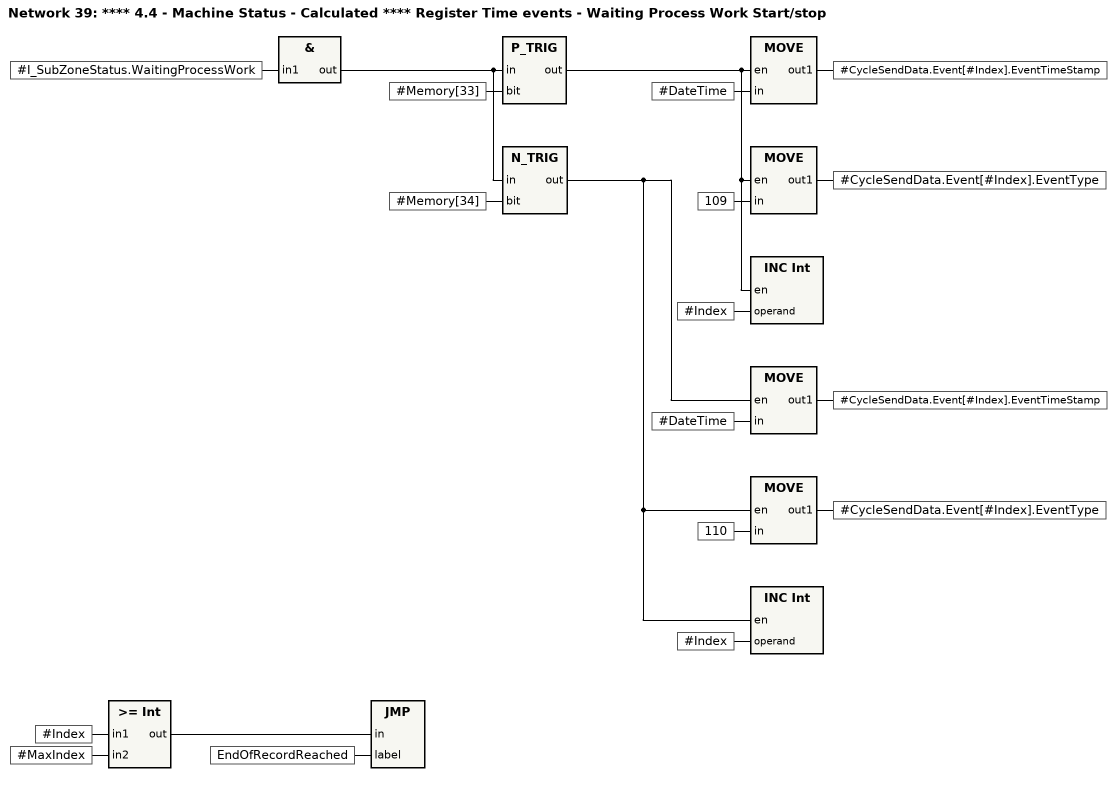
   #_w1 := #I_SubZoneStatus.WaitingProcessWork AND NOT #Memory[33];   // rising edge
   #Memory[33] := #I_SubZoneStatus.WaitingProcessWork;
   IF #_w1 THEN
       #CycleSendData.Event[#Index].EventTimeStamp := #DateTime;
       #CycleSendData.Event[#Index].EventType := 109;
       #Index := #Index + 1;
   END_IF;
   #_w2 := NOT #I_SubZoneStatus.WaitingProcessWork AND #Memory[34];   // falling edge
   #Memory[34] := #I_SubZoneStatus.WaitingProcessWork;
   IF #_w2 THEN
       #CycleSendData.Event[#Index].EventTimeStamp := #DateTime;
       #CycleSendData.Event[#Index].EventType := 110;
       #Index := #Index + 1;
   END_IF;
   IF #Index >= #MaxIndex THEN GOTO EndOfRecordReached; END_IF;
END_REGION

REGION Network 40: **** 4.4 - Machine Status - Calculated **** Register Time events - Process Work Start/stop
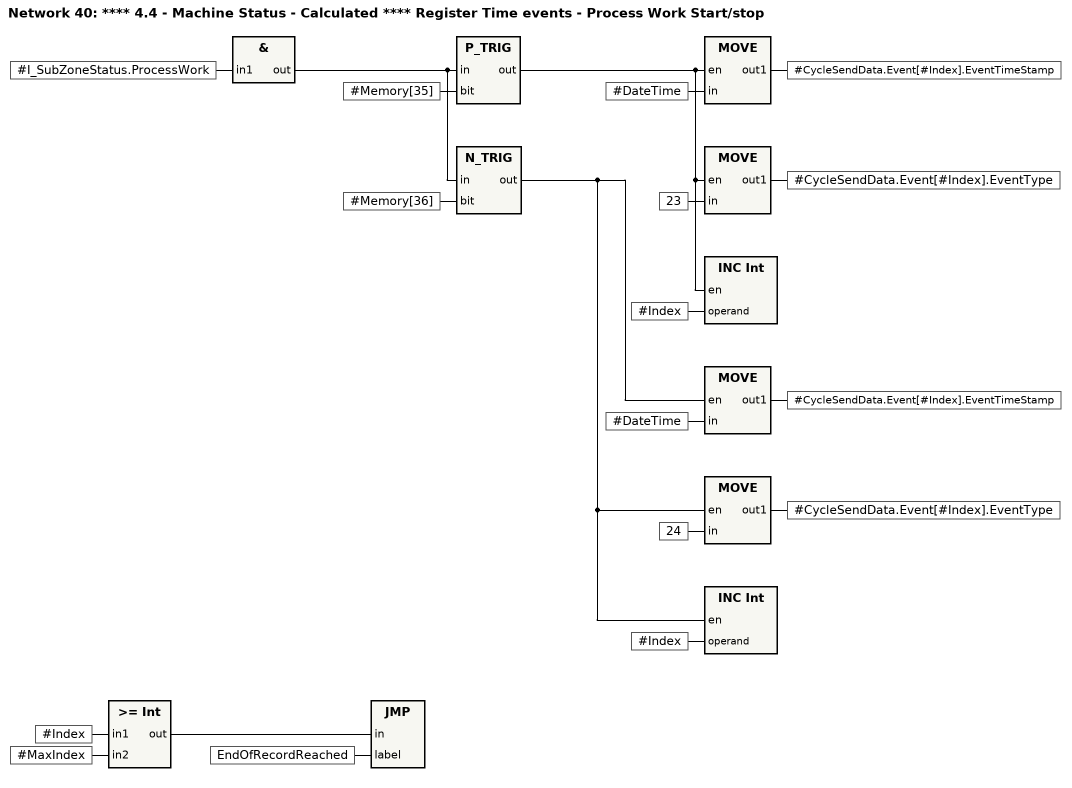
   #_w1 := #I_SubZoneStatus.ProcessWork AND NOT #Memory[35];   // rising edge
   #Memory[35] := #I_SubZoneStatus.ProcessWork;
   IF #_w1 THEN
       #CycleSendData.Event[#Index].EventTimeStamp := #DateTime;
       #CycleSendData.Event[#Index].EventType := 23;
       #Index := #Index + 1;
   END_IF;
   #_w2 := NOT #I_SubZoneStatus.ProcessWork AND #Memory[36];   // falling edge
   #Memory[36] := #I_SubZoneStatus.ProcessWork;
   IF #_w2 THEN
       #CycleSendData.Event[#Index].EventTimeStamp := #DateTime;
       #CycleSendData.Event[#Index].EventType := 24;
       #Index := #Index + 1;
   END_IF;
   IF #Index >= #MaxIndex THEN GOTO EndOfRecordReached; END_IF;
END_REGION

REGION Network 41: **** 4.4 - Machine Status - Calculated **** Register Time events - Cycle Hold
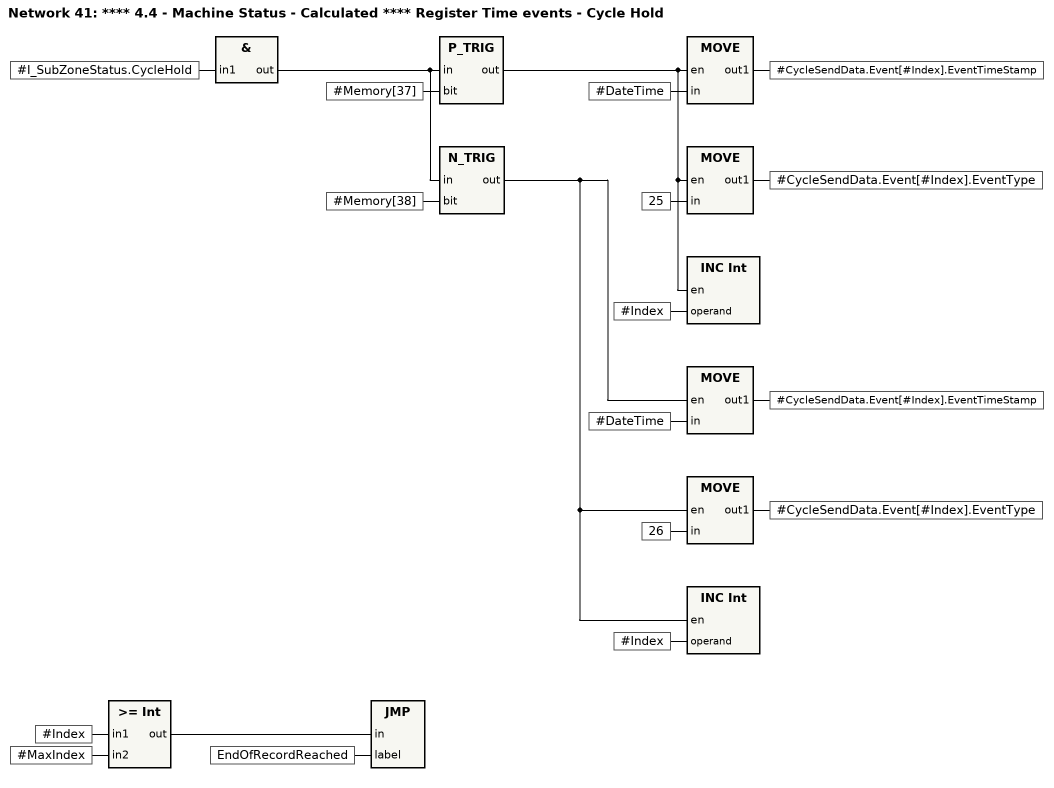
   #_w1 := #I_SubZoneStatus.CycleHold AND NOT #Memory[37];   // rising edge
   #Memory[37] := #I_SubZoneStatus.CycleHold;
   IF #_w1 THEN
       #CycleSendData.Event[#Index].EventTimeStamp := #DateTime;
       #CycleSendData.Event[#Index].EventType := 25;
       #Index := #Index + 1;
   END_IF;
   #_w2 := NOT #I_SubZoneStatus.CycleHold AND #Memory[38];   // falling edge
   #Memory[38] := #I_SubZoneStatus.CycleHold;
   IF #_w2 THEN
       #CycleSendData.Event[#Index].EventTimeStamp := #DateTime;
       #CycleSendData.Event[#Index].EventType := 26;
       #Index := #Index + 1;
   END_IF;
   IF #Index >= #MaxIndex THEN GOTO EndOfRecordReached; END_IF;
END_REGION

REGION Network 42: **** 4.4 - Machine Status - Calculated **** Register Time events - WaitingOutput1 Start/stop
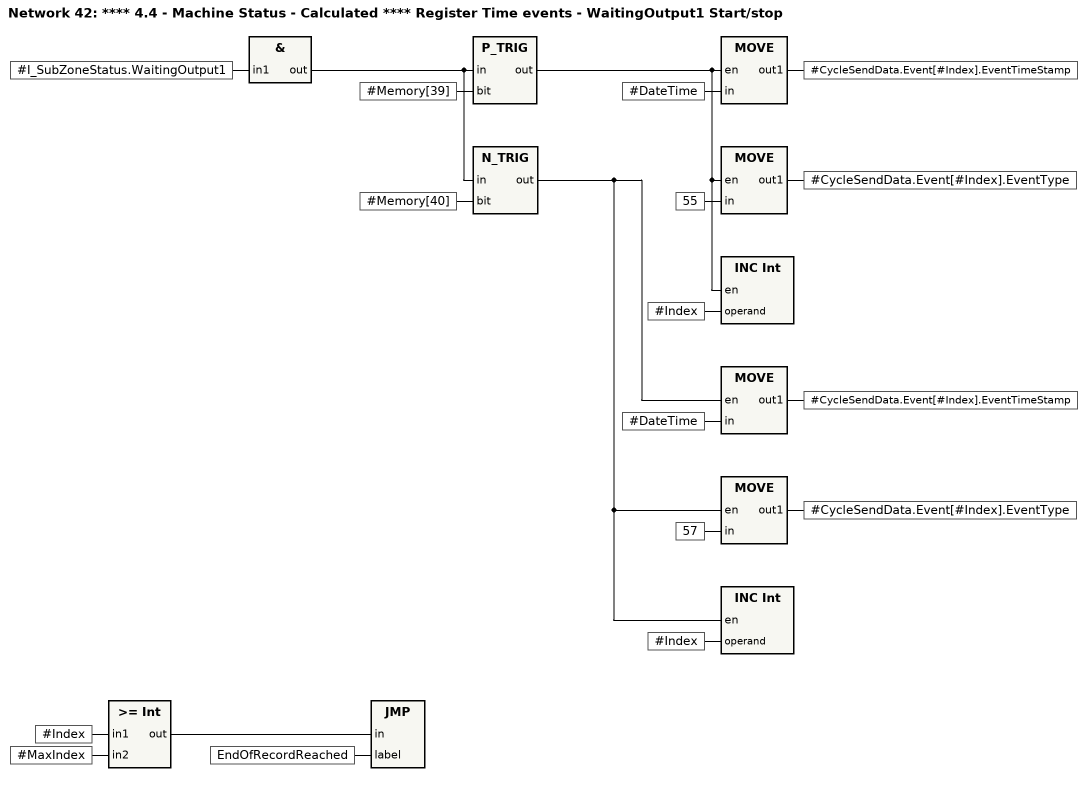
   #_w1 := #I_SubZoneStatus.WaitingOutput1 AND NOT #Memory[39];   // rising edge
   #Memory[39] := #I_SubZoneStatus.WaitingOutput1;
   IF #_w1 THEN
       #CycleSendData.Event[#Index].EventTimeStamp := #DateTime;
       #CycleSendData.Event[#Index].EventType := 55;
       #Index := #Index + 1;
   END_IF;
   #_w2 := NOT #I_SubZoneStatus.WaitingOutput1 AND #Memory[40];   // falling edge
   #Memory[40] := #I_SubZoneStatus.WaitingOutput1;
   IF #_w2 THEN
       #CycleSendData.Event[#Index].EventTimeStamp := #DateTime;
       #CycleSendData.Event[#Index].EventType := 57;
       #Index := #Index + 1;
   END_IF;
   IF #Index >= #MaxIndex THEN GOTO EndOfRecordReached; END_IF;
END_REGION

REGION Network 43: **** 4.4 - Machine Status - Calculated **** Register Time events - WaitingOutput2 Start/stop
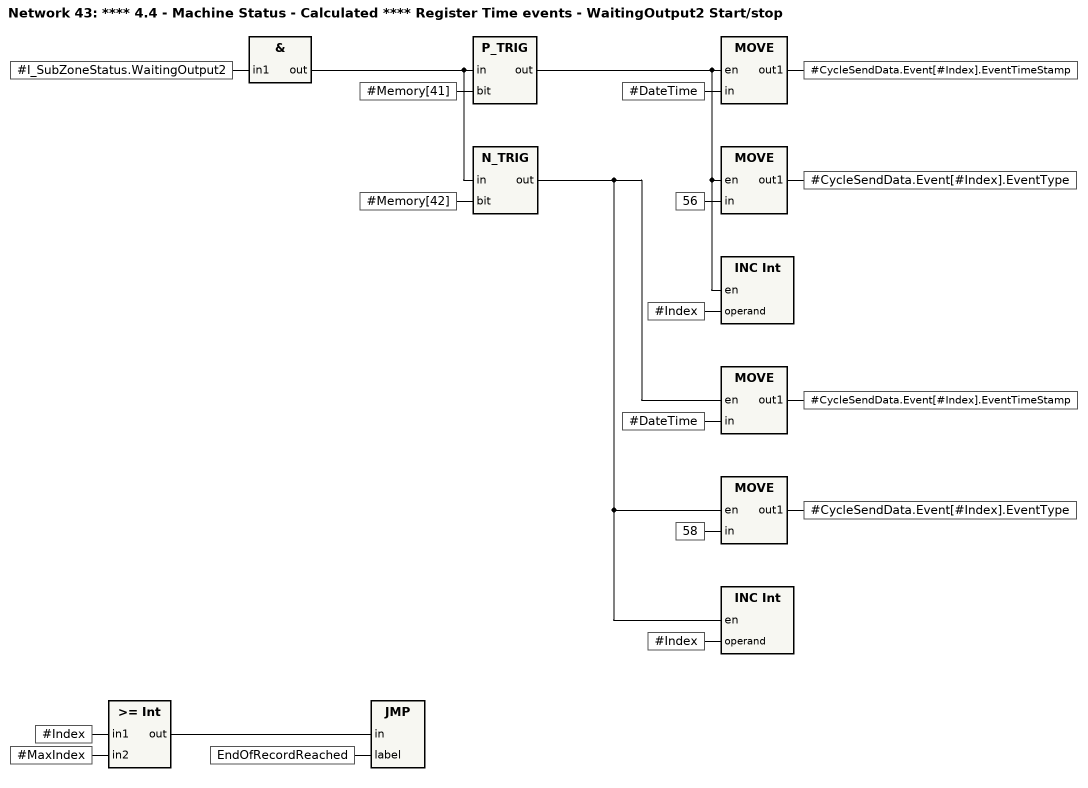
   #_w1 := #I_SubZoneStatus.WaitingOutput2 AND NOT #Memory[41];   // rising edge
   #Memory[41] := #I_SubZoneStatus.WaitingOutput2;
   IF #_w1 THEN
       #CycleSendData.Event[#Index].EventTimeStamp := #DateTime;
       #CycleSendData.Event[#Index].EventType := 56;
       #Index := #Index + 1;
   END_IF;
   #_w2 := NOT #I_SubZoneStatus.WaitingOutput2 AND #Memory[42];   // falling edge
   #Memory[42] := #I_SubZoneStatus.WaitingOutput2;
   IF #_w2 THEN
       #CycleSendData.Event[#Index].EventTimeStamp := #DateTime;
       #CycleSendData.Event[#Index].EventType := 58;
       #Index := #Index + 1;
   END_IF;
   IF #Index >= #MaxIndex THEN GOTO EndOfRecordReached; END_IF;
END_REGION

REGION Network 44: **** 4.4 - Machine Status - Calculated **** Register Time events - Outfeed1 Start/stop
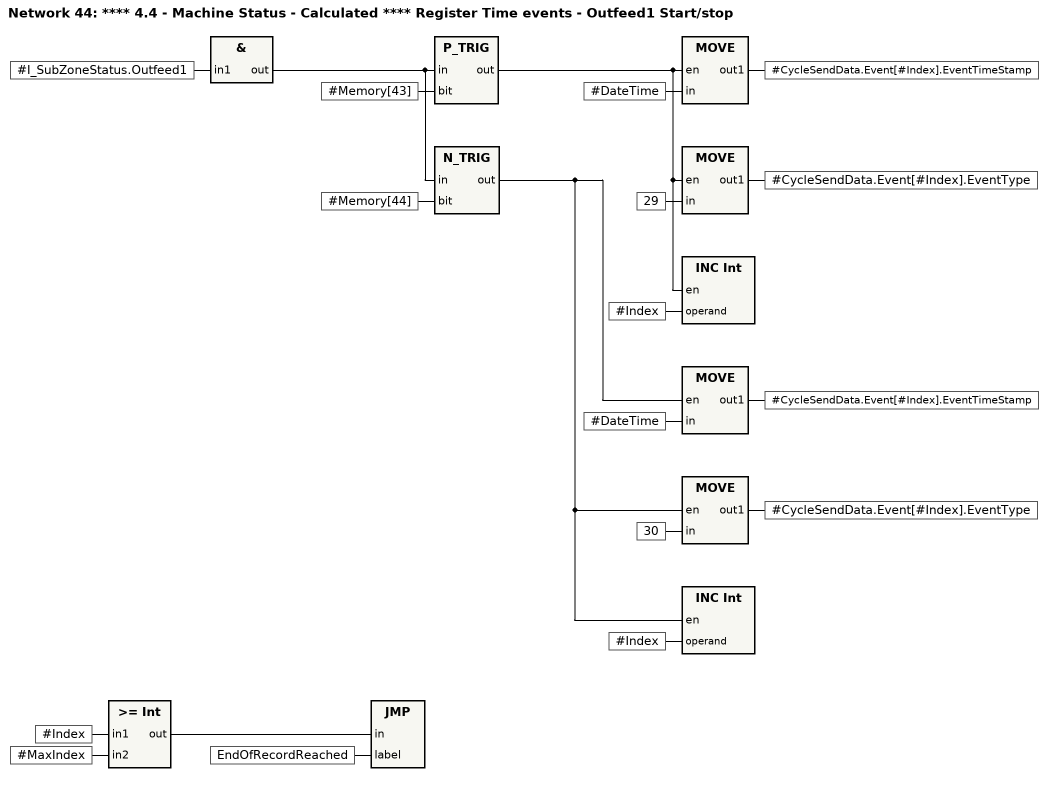
   #_w1 := #I_SubZoneStatus.Outfeed1 AND NOT #Memory[43];   // rising edge
   #Memory[43] := #I_SubZoneStatus.Outfeed1;
   IF #_w1 THEN
       #CycleSendData.Event[#Index].EventTimeStamp := #DateTime;
       #CycleSendData.Event[#Index].EventType := 29;
       #Index := #Index + 1;
   END_IF;
   #_w2 := NOT #I_SubZoneStatus.Outfeed1 AND #Memory[44];   // falling edge
   #Memory[44] := #I_SubZoneStatus.Outfeed1;
   IF #_w2 THEN
       #CycleSendData.Event[#Index].EventTimeStamp := #DateTime;
       #CycleSendData.Event[#Index].EventType := 30;
       #Index := #Index + 1;
   END_IF;
   IF #Index >= #MaxIndex THEN GOTO EndOfRecordReached; END_IF;
END_REGION

REGION Network 45: **** 4.4 - Machine Status - Calculated **** Register Time events - Outfeed2 Start/stop
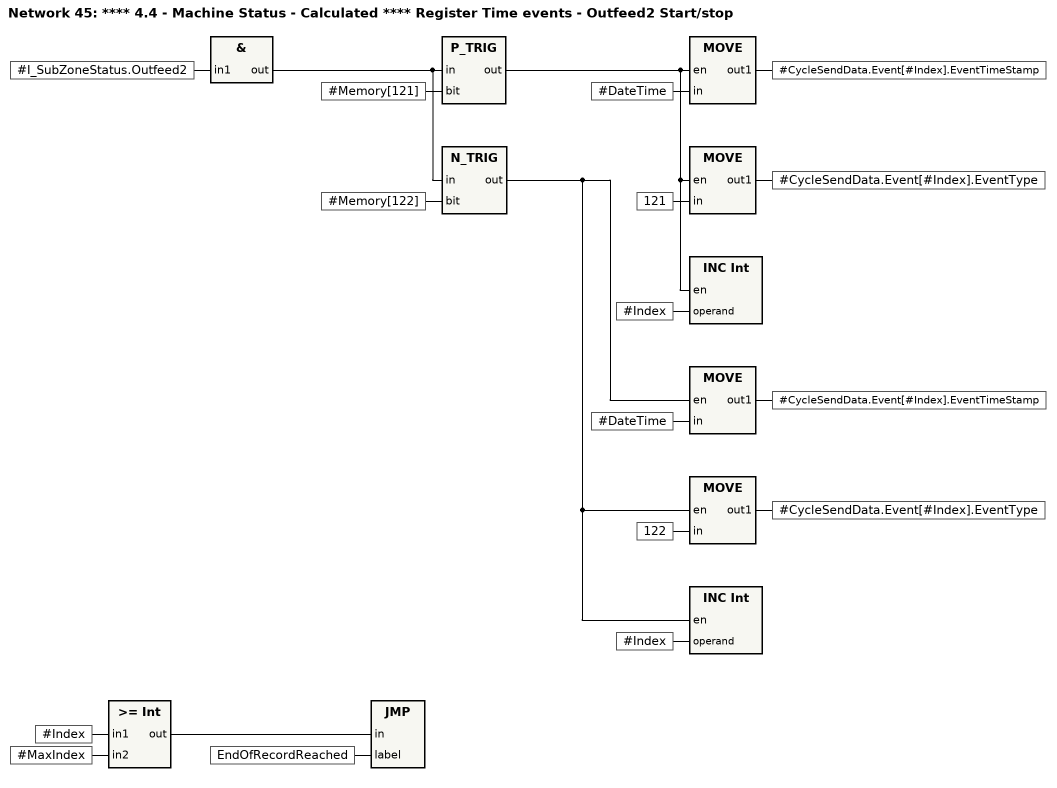
   #_w1 := #I_SubZoneStatus.Outfeed2 AND NOT #Memory[121];   // rising edge
   #Memory[121] := #I_SubZoneStatus.Outfeed2;
   IF #_w1 THEN
       #CycleSendData.Event[#Index].EventTimeStamp := #DateTime;
       #CycleSendData.Event[#Index].EventType := 121;
       #Index := #Index + 1;
   END_IF;
   #_w2 := NOT #I_SubZoneStatus.Outfeed2 AND #Memory[122];   // falling edge
   #Memory[122] := #I_SubZoneStatus.Outfeed2;
   IF #_w2 THEN
       #CycleSendData.Event[#Index].EventTimeStamp := #DateTime;
       #CycleSendData.Event[#Index].EventType := 122;
       #Index := #Index + 1;
   END_IF;
   IF #Index >= #MaxIndex THEN GOTO EndOfRecordReached; END_IF;
END_REGION

REGION Network 46: **** 4.4 - Machine Status - Calculated **** Register Time events - Recovery Time Start/stop
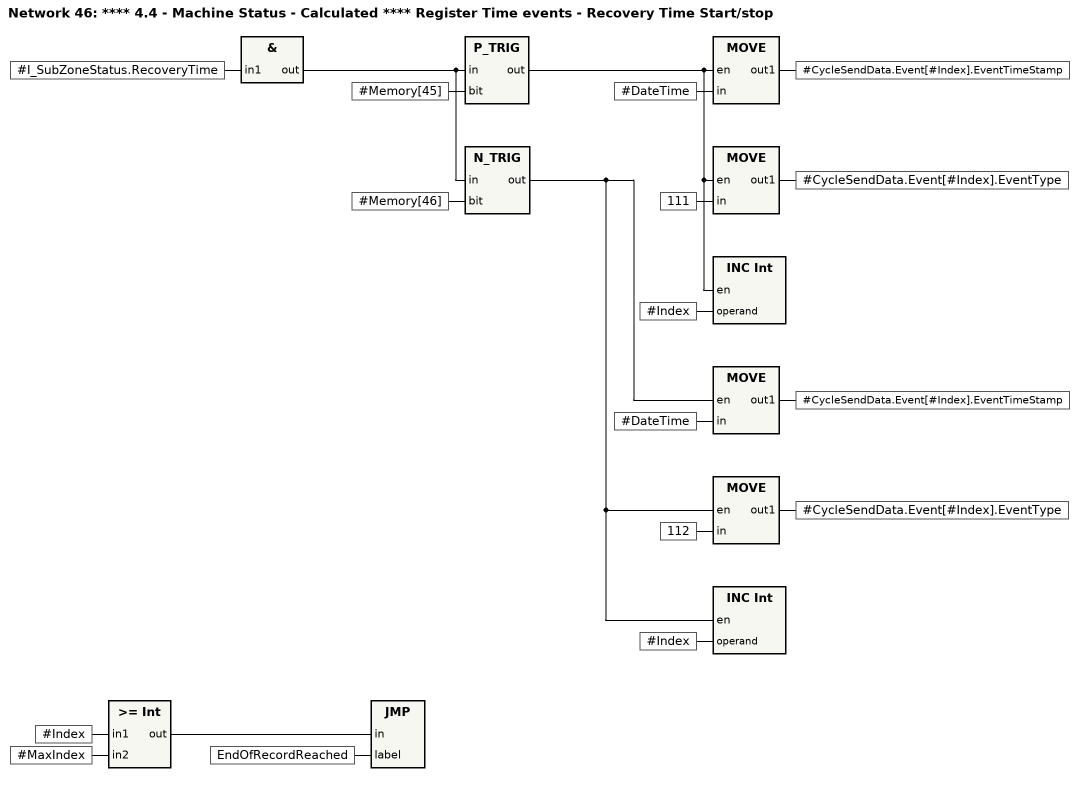
   #_w1 := #I_SubZoneStatus.RecoveryTime AND NOT #Memory[45];   // rising edge
   #Memory[45] := #I_SubZoneStatus.RecoveryTime;
   IF #_w1 THEN
       #CycleSendData.Event[#Index].EventTimeStamp := #DateTime;
       #CycleSendData.Event[#Index].EventType := 111;
       #Index := #Index + 1;
   END_IF;
   #_w2 := NOT #I_SubZoneStatus.RecoveryTime AND #Memory[46];   // falling edge
   #Memory[46] := #I_SubZoneStatus.RecoveryTime;
   IF #_w2 THEN
       #CycleSendData.Event[#Index].EventTimeStamp := #DateTime;
       #CycleSendData.Event[#Index].EventType := 112;
       #Index := #Index + 1;
   END_IF;
   IF #Index >= #MaxIndex THEN GOTO EndOfRecordReached; END_IF;
END_REGION

REGION Network 47: **** 4.4 - Machine Status - Calculated **** Register Time events - QualityNok Start/stop
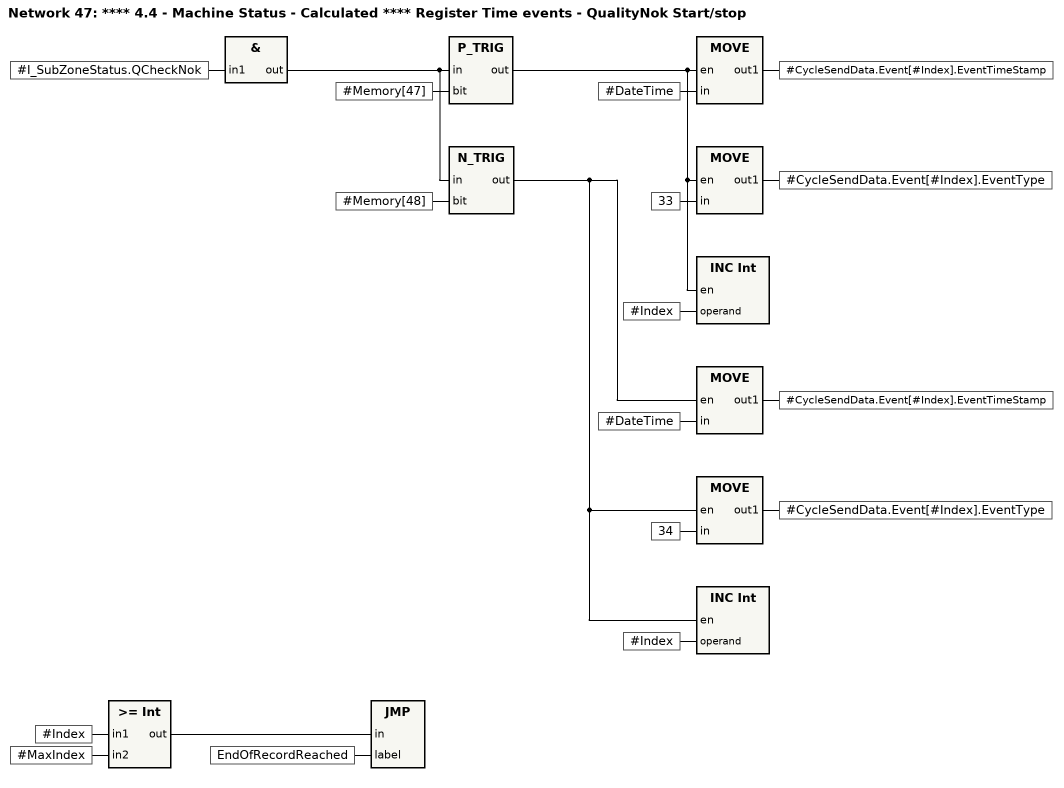
   #_w1 := #I_SubZoneStatus.QCheckNok AND NOT #Memory[47];   // rising edge
   #Memory[47] := #I_SubZoneStatus.QCheckNok;
   IF #_w1 THEN
       #CycleSendData.Event[#Index].EventTimeStamp := #DateTime;
       #CycleSendData.Event[#Index].EventType := 33;
       #Index := #Index + 1;
   END_IF;
   #_w2 := NOT #I_SubZoneStatus.QCheckNok AND #Memory[48];   // falling edge
   #Memory[48] := #I_SubZoneStatus.QCheckNok;
   IF #_w2 THEN
       #CycleSendData.Event[#Index].EventTimeStamp := #DateTime;
       #CycleSendData.Event[#Index].EventType := 34;
       #Index := #Index + 1;
   END_IF;
   IF #Index >= #MaxIndex THEN GOTO EndOfRecordReached; END_IF;
END_REGION

REGION Network 48: **** 4.4 - Machine Status - Calculated **** Register Time events - Bypass Start/stop
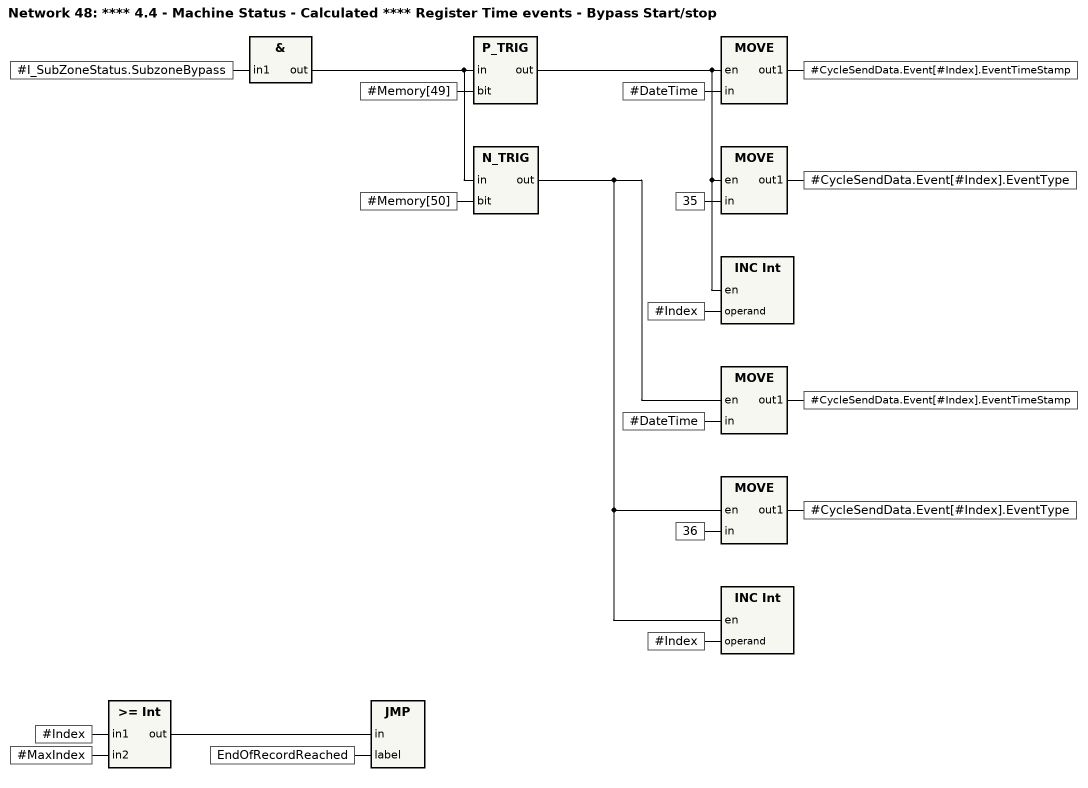
   #_w1 := #I_SubZoneStatus.SubzoneBypass AND NOT #Memory[49];   // rising edge
   #Memory[49] := #I_SubZoneStatus.SubzoneBypass;
   IF #_w1 THEN
       #CycleSendData.Event[#Index].EventTimeStamp := #DateTime;
       #CycleSendData.Event[#Index].EventType := 35;
       #Index := #Index + 1;
   END_IF;
   #_w2 := NOT #I_SubZoneStatus.SubzoneBypass AND #Memory[50];   // falling edge
   #Memory[50] := #I_SubZoneStatus.SubzoneBypass;
   IF #_w2 THEN
       #CycleSendData.Event[#Index].EventTimeStamp := #DateTime;
       #CycleSendData.Event[#Index].EventType := 36;
       #Index := #Index + 1;
   END_IF;
   IF #Index >= #MaxIndex THEN GOTO EndOfRecordReached; END_IF;
END_REGION

REGION Network 49: **** 4.4 - Machine Status - Calculated **** Register Time events - Manual Start/stop
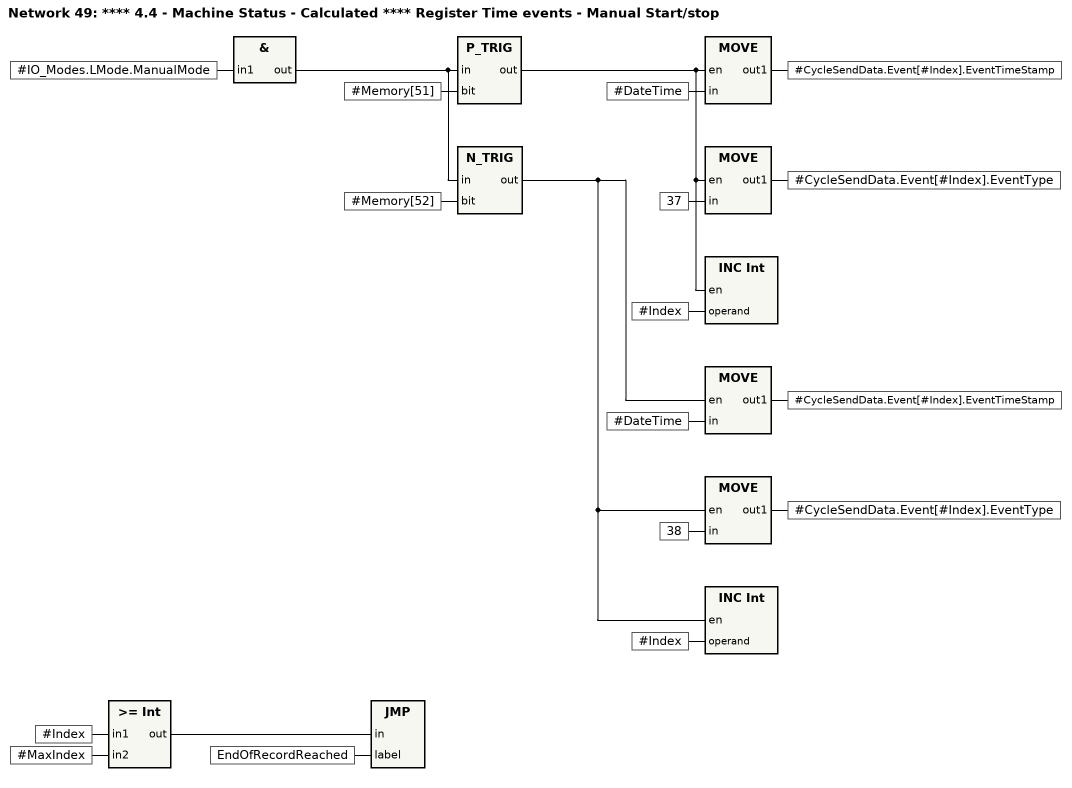
   #_w1 := #IO_Modes.LMode.ManualMode AND NOT #Memory[51];   // rising edge
   #Memory[51] := #IO_Modes.LMode.ManualMode;
   IF #_w1 THEN
       #CycleSendData.Event[#Index].EventTimeStamp := #DateTime;
       #CycleSendData.Event[#Index].EventType := 37;
       #Index := #Index + 1;
   END_IF;
   #_w2 := NOT #IO_Modes.LMode.ManualMode AND #Memory[52];   // falling edge
   #Memory[52] := #IO_Modes.LMode.ManualMode;
   IF #_w2 THEN
       #CycleSendData.Event[#Index].EventTimeStamp := #DateTime;
       #CycleSendData.Event[#Index].EventType := 38;
       #Index := #Index + 1;
   END_IF;
   IF #Index >= #MaxIndex THEN GOTO EndOfRecordReached; END_IF;
END_REGION

REGION Network 50: **** 4.4 - Machine Status - Calculated **** Register Time events - CycleStop Start/stop
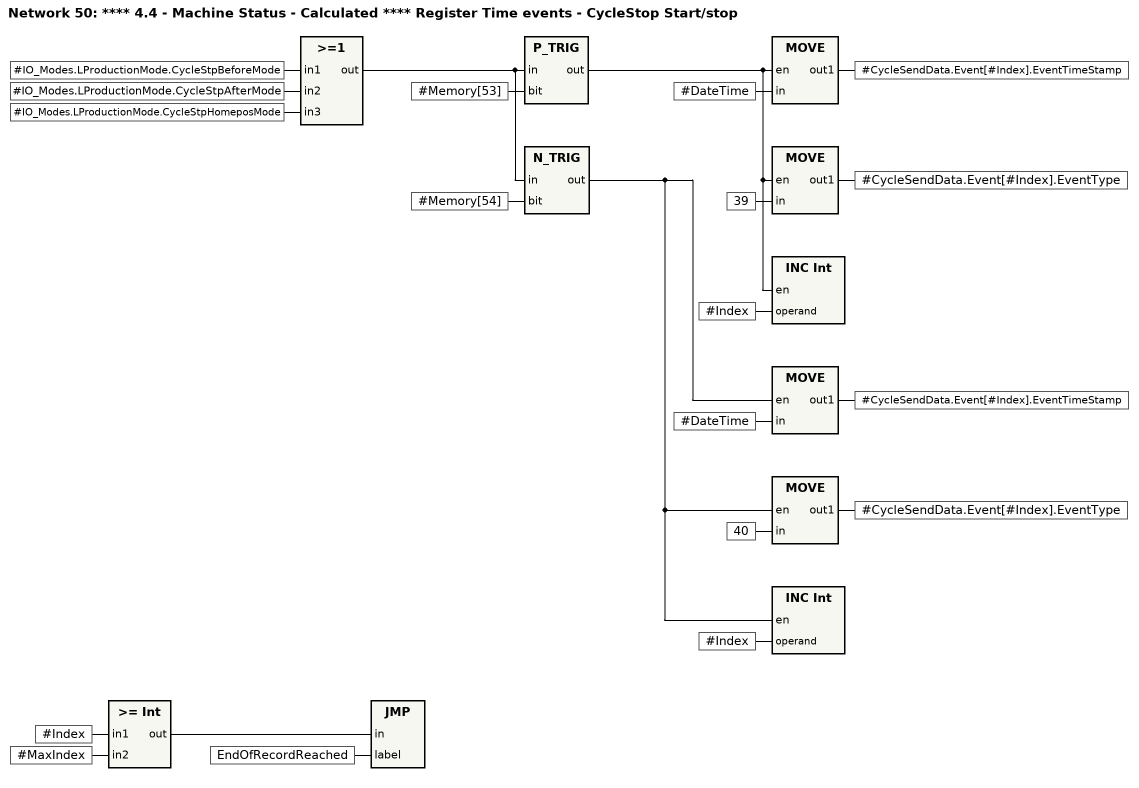
   #_w1 := #IO_Modes.LProductionMode.CycleStpBeforeMode OR #IO_Modes.LProductionMode.CycleStpAfterMode OR #IO_Modes.LProductionMode.CycleStpHomeposMode;
   #_w2 := #_w1 AND NOT #Memory[53];   // rising edge
   #Memory[53] := #_w1;
   IF #_w2 THEN
       #CycleSendData.Event[#Index].EventTimeStamp := #DateTime;
       #CycleSendData.Event[#Index].EventType := 39;
       #Index := #Index + 1;
   END_IF;
   #_w3 := NOT #_w1 AND #Memory[54];   // falling edge
   #Memory[54] := #_w1;
   IF #_w3 THEN
       #CycleSendData.Event[#Index].EventTimeStamp := #DateTime;
       #CycleSendData.Event[#Index].EventType := 40;
       #Index := #Index + 1;
   END_IF;
   IF #Index >= #MaxIndex THEN GOTO EndOfRecordReached; END_IF;
END_REGION

REGION Network 51: **** 4.4 - Machine Status - Calculated **** Register Time events - SimulationMode Start/stop
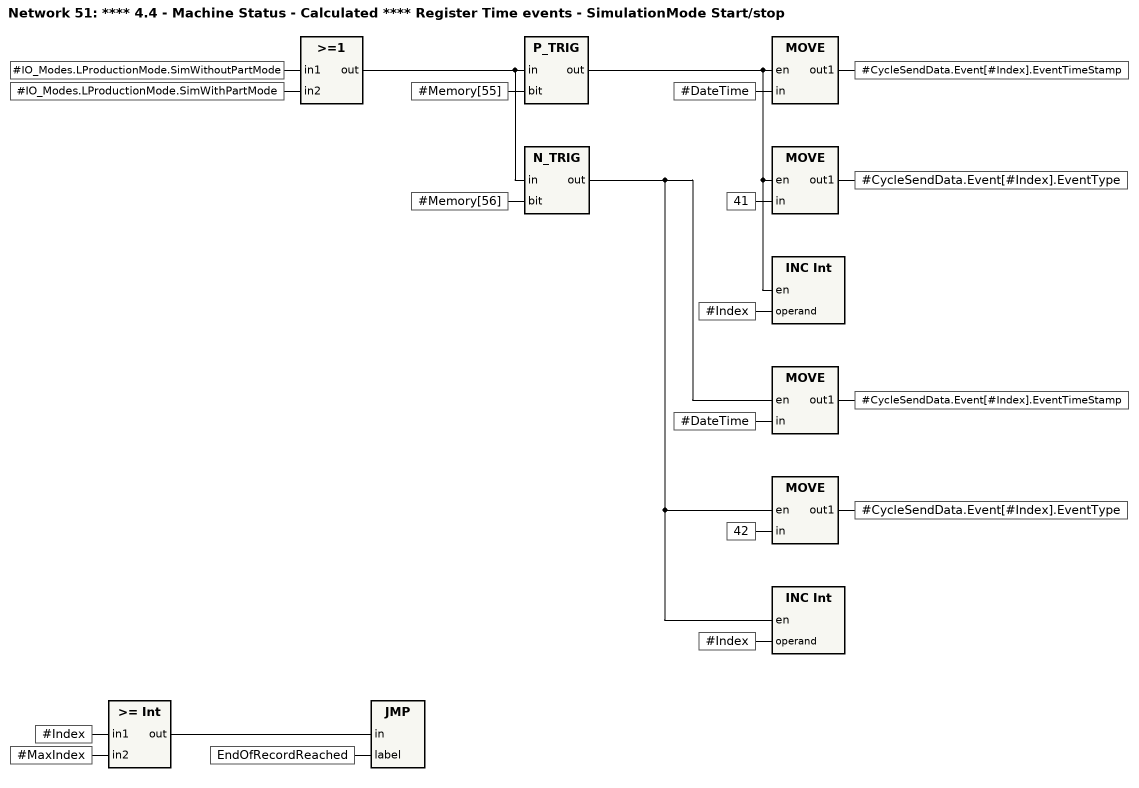
   #_w1 := #IO_Modes.LProductionMode.SimWithoutPartMode OR #IO_Modes.LProductionMode.SimWithPartMode;
   #_w2 := #_w1 AND NOT #Memory[55];   // rising edge
   #Memory[55] := #_w1;
   IF #_w2 THEN
       #CycleSendData.Event[#Index].EventTimeStamp := #DateTime;
       #CycleSendData.Event[#Index].EventType := 41;
       #Index := #Index + 1;
   END_IF;
   #_w3 := NOT #_w1 AND #Memory[56];   // falling edge
   #Memory[56] := #_w1;
   IF #_w3 THEN
       #CycleSendData.Event[#Index].EventTimeStamp := #DateTime;
       #CycleSendData.Event[#Index].EventType := 42;
       #Index := #Index + 1;
   END_IF;
   IF #Index >= #MaxIndex THEN GOTO EndOfRecordReached; END_IF;
END_REGION

REGION Network 52: **** 4.4 - Machine Status - Calculated **** Register Time events - EmptyStation Start/stop
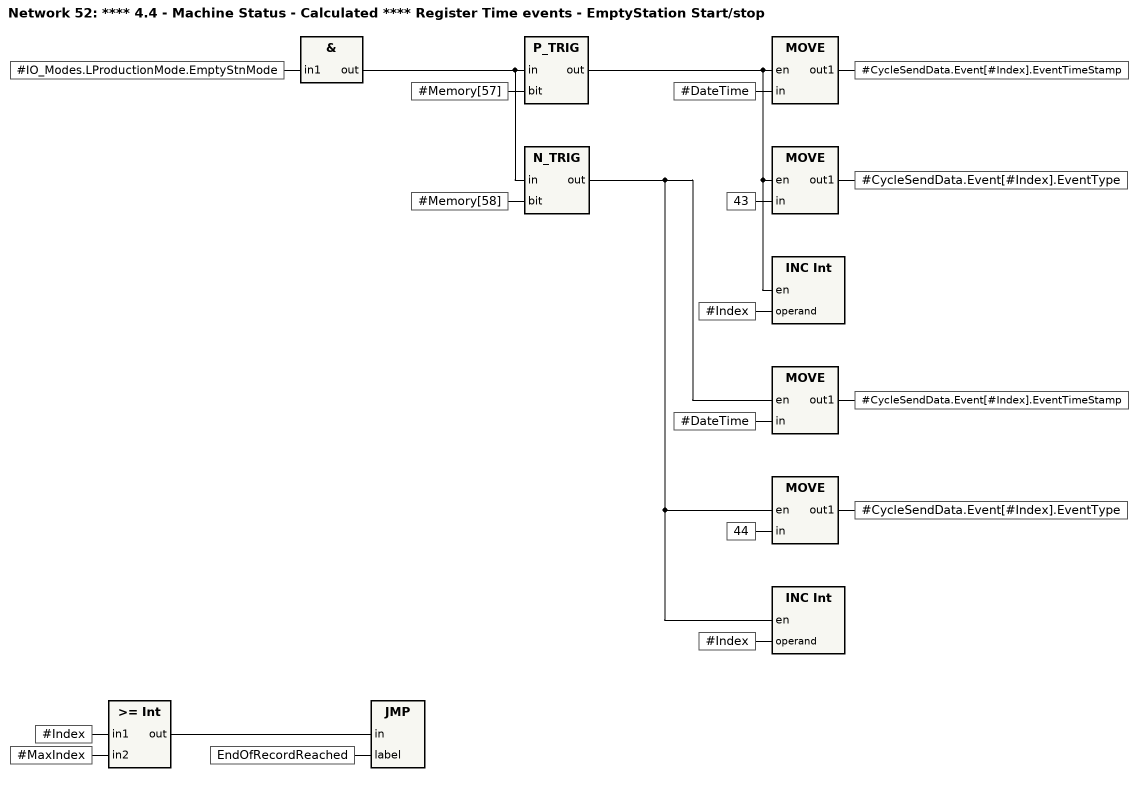
   #_w1 := #IO_Modes.LProductionMode.EmptyStnMode AND NOT #Memory[57];   // rising edge
   #Memory[57] := #IO_Modes.LProductionMode.EmptyStnMode;
   IF #_w1 THEN
       #CycleSendData.Event[#Index].EventTimeStamp := #DateTime;
       #CycleSendData.Event[#Index].EventType := 43;
       #Index := #Index + 1;
   END_IF;
   #_w2 := NOT #IO_Modes.LProductionMode.EmptyStnMode AND #Memory[58];   // falling edge
   #Memory[58] := #IO_Modes.LProductionMode.EmptyStnMode;
   IF #_w2 THEN
       #CycleSendData.Event[#Index].EventTimeStamp := #DateTime;
       #CycleSendData.Event[#Index].EventType := 44;
       #Index := #Index + 1;
   END_IF;
   IF #Index >= #MaxIndex THEN GOTO EndOfRecordReached; END_IF;
END_REGION

REGION Network 53: **** 4.4 - Machine Status - Calculated **** Register Time events - OperatorWork1 Start/stop
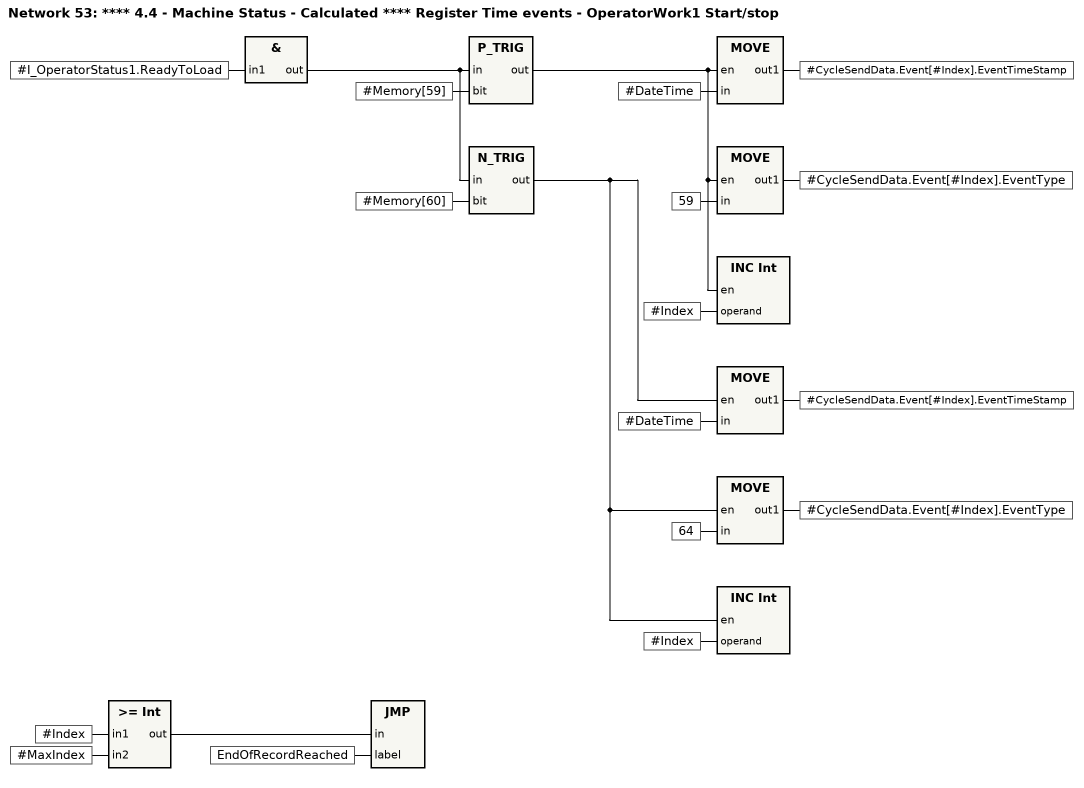
   #_w1 := #I_OperatorStatus1.ReadyToLoad AND NOT #Memory[59];   // rising edge
   #Memory[59] := #I_OperatorStatus1.ReadyToLoad;
   IF #_w1 THEN
       #CycleSendData.Event[#Index].EventTimeStamp := #DateTime;
       #CycleSendData.Event[#Index].EventType := 59;
       #Index := #Index + 1;
   END_IF;
   #_w2 := NOT #I_OperatorStatus1.ReadyToLoad AND #Memory[60];   // falling edge
   #Memory[60] := #I_OperatorStatus1.ReadyToLoad;
   IF #_w2 THEN
       #CycleSendData.Event[#Index].EventTimeStamp := #DateTime;
       #CycleSendData.Event[#Index].EventType := 64;
       #Index := #Index + 1;
   END_IF;
   IF #Index >= #MaxIndex THEN GOTO EndOfRecordReached; END_IF;
END_REGION

REGION Network 54: **** 4.4 - Machine Status - Calculated **** Register Time events - OperatorWork2 Start/stop
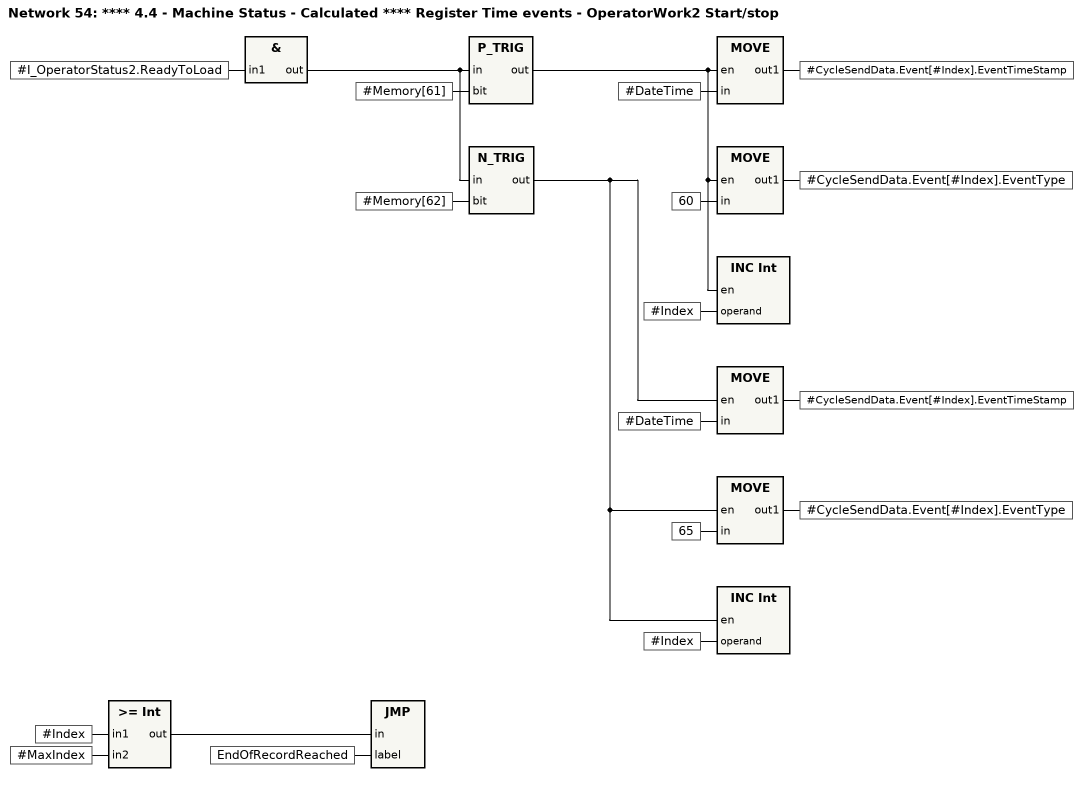
   #_w1 := #I_OperatorStatus2.ReadyToLoad AND NOT #Memory[61];   // rising edge
   #Memory[61] := #I_OperatorStatus2.ReadyToLoad;
   IF #_w1 THEN
       #CycleSendData.Event[#Index].EventTimeStamp := #DateTime;
       #CycleSendData.Event[#Index].EventType := 60;
       #Index := #Index + 1;
   END_IF;
   #_w2 := NOT #I_OperatorStatus2.ReadyToLoad AND #Memory[62];   // falling edge
   #Memory[62] := #I_OperatorStatus2.ReadyToLoad;
   IF #_w2 THEN
       #CycleSendData.Event[#Index].EventTimeStamp := #DateTime;
       #CycleSendData.Event[#Index].EventType := 65;
       #Index := #Index + 1;
   END_IF;
   IF #Index >= #MaxIndex THEN GOTO EndOfRecordReached; END_IF;
END_REGION

REGION Network 55: **** 4.4 - Machine Status - Calculated **** Register Time events - OperatorWork3 Start/stop
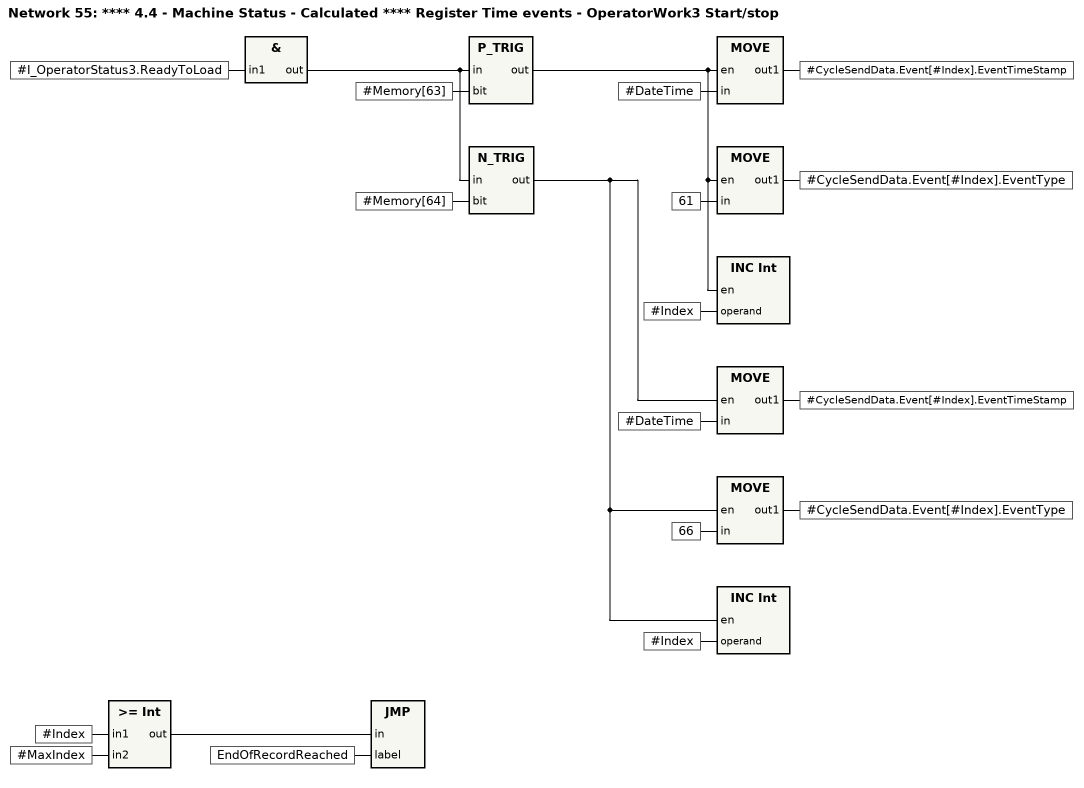
   #_w1 := #I_OperatorStatus3.ReadyToLoad AND NOT #Memory[63];   // rising edge
   #Memory[63] := #I_OperatorStatus3.ReadyToLoad;
   IF #_w1 THEN
       #CycleSendData.Event[#Index].EventTimeStamp := #DateTime;
       #CycleSendData.Event[#Index].EventType := 61;
       #Index := #Index + 1;
   END_IF;
   #_w2 := NOT #I_OperatorStatus3.ReadyToLoad AND #Memory[64];   // falling edge
   #Memory[64] := #I_OperatorStatus3.ReadyToLoad;
   IF #_w2 THEN
       #CycleSendData.Event[#Index].EventTimeStamp := #DateTime;
       #CycleSendData.Event[#Index].EventType := 66;
       #Index := #Index + 1;
   END_IF;
   IF #Index >= #MaxIndex THEN GOTO EndOfRecordReached; END_IF;
END_REGION

REGION Network 56: **** 4.4 - Machine Status - Calculated **** Register Time events - OperatorWork4 Start/stop
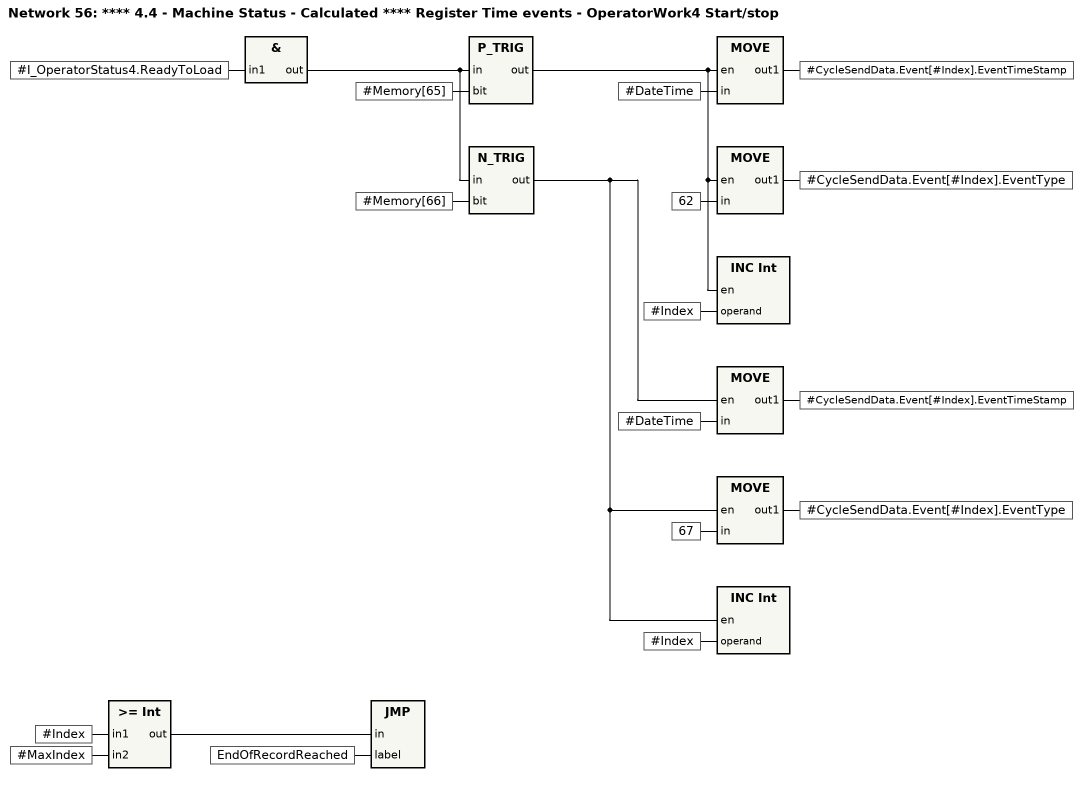
   #_w1 := #I_OperatorStatus4.ReadyToLoad AND NOT #Memory[65];   // rising edge
   #Memory[65] := #I_OperatorStatus4.ReadyToLoad;
   IF #_w1 THEN
       #CycleSendData.Event[#Index].EventTimeStamp := #DateTime;
       #CycleSendData.Event[#Index].EventType := 62;
       #Index := #Index + 1;
   END_IF;
   #_w2 := NOT #I_OperatorStatus4.ReadyToLoad AND #Memory[66];   // falling edge
   #Memory[66] := #I_OperatorStatus4.ReadyToLoad;
   IF #_w2 THEN
       #CycleSendData.Event[#Index].EventTimeStamp := #DateTime;
       #CycleSendData.Event[#Index].EventType := 67;
       #Index := #Index + 1;
   END_IF;
   IF #Index >= #MaxIndex THEN GOTO EndOfRecordReached; END_IF;
END_REGION

REGION Network 57: **** 4.4 - Machine Status - Calculated **** Register Time events - OperatorWork5 Start/stop
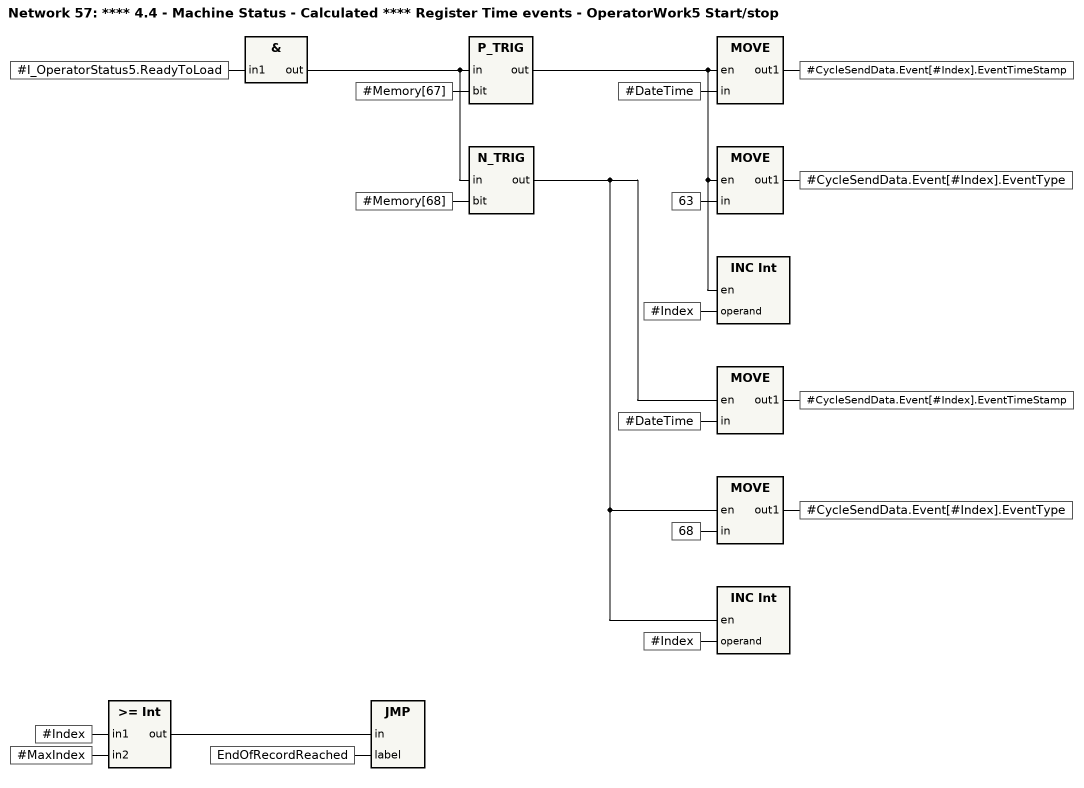
   #_w1 := #I_OperatorStatus5.ReadyToLoad AND NOT #Memory[67];   // rising edge
   #Memory[67] := #I_OperatorStatus5.ReadyToLoad;
   IF #_w1 THEN
       #CycleSendData.Event[#Index].EventTimeStamp := #DateTime;
       #CycleSendData.Event[#Index].EventType := 63;
       #Index := #Index + 1;
   END_IF;
   #_w2 := NOT #I_OperatorStatus5.ReadyToLoad AND #Memory[68];   // falling edge
   #Memory[68] := #I_OperatorStatus5.ReadyToLoad;
   IF #_w2 THEN
       #CycleSendData.Event[#Index].EventTimeStamp := #DateTime;
       #CycleSendData.Event[#Index].EventType := 68;
       #Index := #Index + 1;
   END_IF;
   IF #Index >= #MaxIndex THEN GOTO EndOfRecordReached; END_IF;
END_REGION

REGION Network 58: **** 4.4 - Machine Status - Calculated **** Register Time events - OperatorOverCycle1 Start/stop
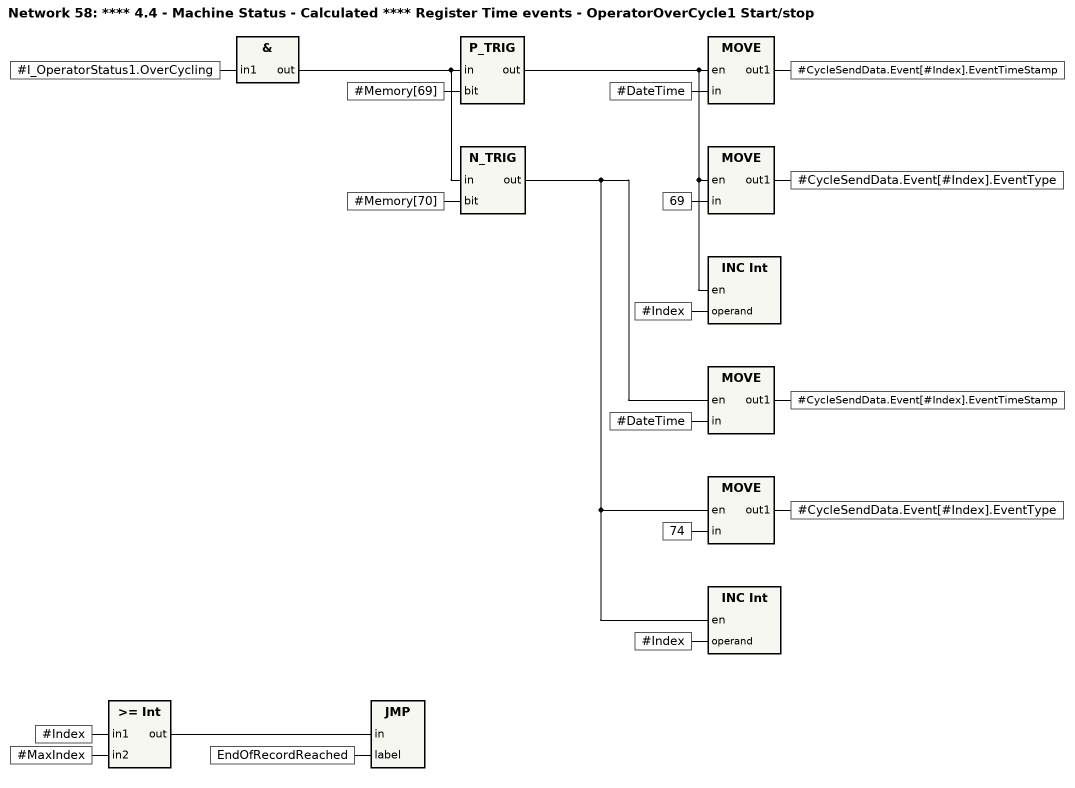
   #_w1 := #I_OperatorStatus1.OverCycling AND NOT #Memory[69];   // rising edge
   #Memory[69] := #I_OperatorStatus1.OverCycling;
   IF #_w1 THEN
       #CycleSendData.Event[#Index].EventTimeStamp := #DateTime;
       #CycleSendData.Event[#Index].EventType := 69;
       #Index := #Index + 1;
   END_IF;
   #_w2 := NOT #I_OperatorStatus1.OverCycling AND #Memory[70];   // falling edge
   #Memory[70] := #I_OperatorStatus1.OverCycling;
   IF #_w2 THEN
       #CycleSendData.Event[#Index].EventTimeStamp := #DateTime;
       #CycleSendData.Event[#Index].EventType := 74;
       #Index := #Index + 1;
   END_IF;
   IF #Index >= #MaxIndex THEN GOTO EndOfRecordReached; END_IF;
END_REGION

REGION Network 59: **** 4.4 - Machine Status - Calculated **** Register Time events - OperatorOverCycle2 Start/stop
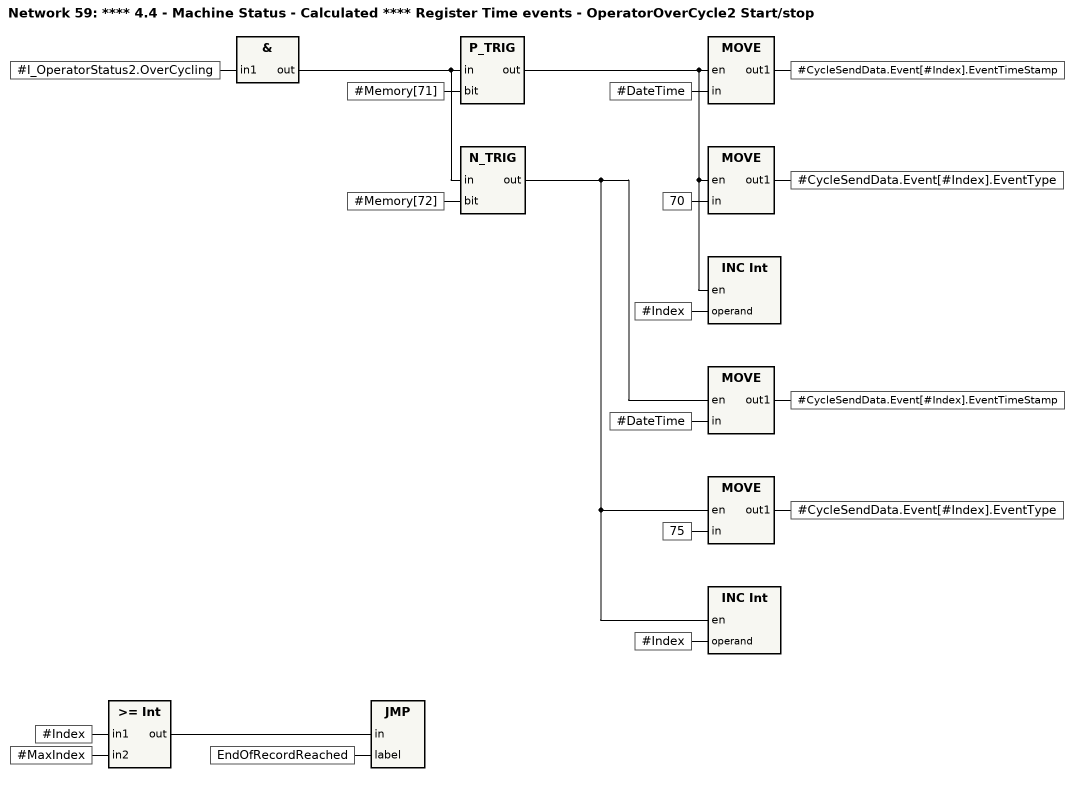
   #_w1 := #I_OperatorStatus2.OverCycling AND NOT #Memory[71];   // rising edge
   #Memory[71] := #I_OperatorStatus2.OverCycling;
   IF #_w1 THEN
       #CycleSendData.Event[#Index].EventTimeStamp := #DateTime;
       #CycleSendData.Event[#Index].EventType := 70;
       #Index := #Index + 1;
   END_IF;
   #_w2 := NOT #I_OperatorStatus2.OverCycling AND #Memory[72];   // falling edge
   #Memory[72] := #I_OperatorStatus2.OverCycling;
   IF #_w2 THEN
       #CycleSendData.Event[#Index].EventTimeStamp := #DateTime;
       #CycleSendData.Event[#Index].EventType := 75;
       #Index := #Index + 1;
   END_IF;
   IF #Index >= #MaxIndex THEN GOTO EndOfRecordReached; END_IF;
END_REGION

REGION Network 60: **** 4.4 - Machine Status - Calculated **** Register Time events - OperatorOverCycle3 Start/stop
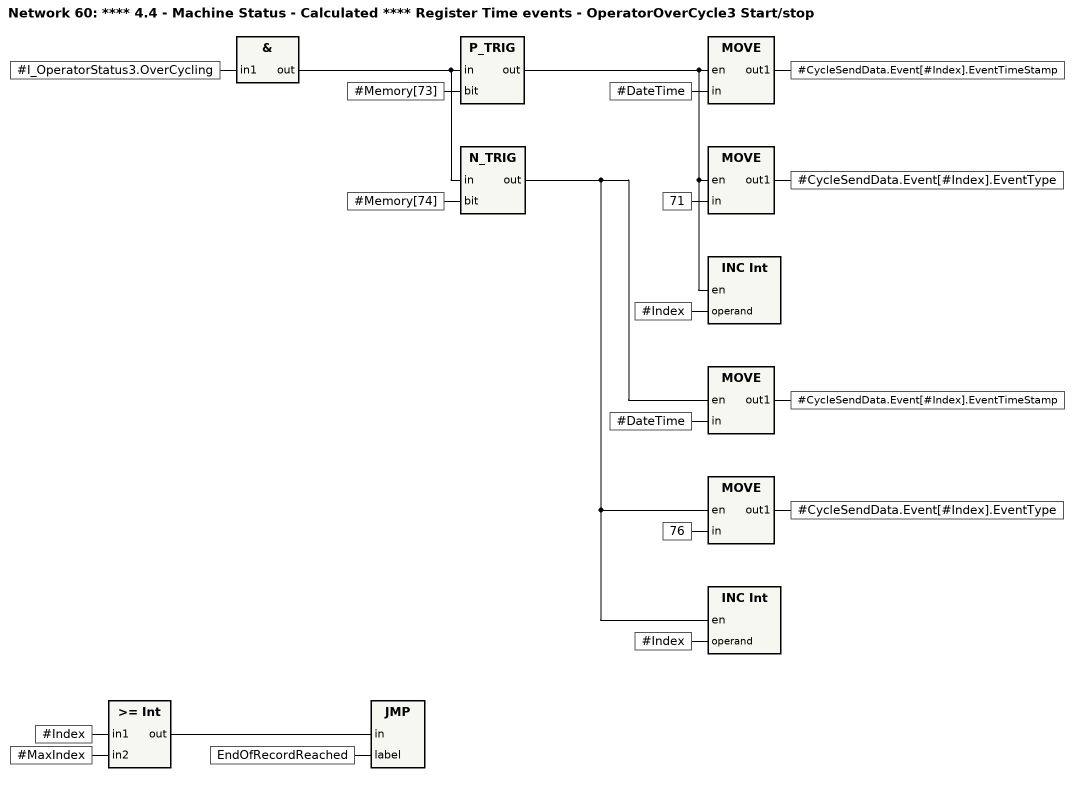
   #_w1 := #I_OperatorStatus3.OverCycling AND NOT #Memory[73];   // rising edge
   #Memory[73] := #I_OperatorStatus3.OverCycling;
   IF #_w1 THEN
       #CycleSendData.Event[#Index].EventTimeStamp := #DateTime;
       #CycleSendData.Event[#Index].EventType := 71;
       #Index := #Index + 1;
   END_IF;
   #_w2 := NOT #I_OperatorStatus3.OverCycling AND #Memory[74];   // falling edge
   #Memory[74] := #I_OperatorStatus3.OverCycling;
   IF #_w2 THEN
       #CycleSendData.Event[#Index].EventTimeStamp := #DateTime;
       #CycleSendData.Event[#Index].EventType := 76;
       #Index := #Index + 1;
   END_IF;
   IF #Index >= #MaxIndex THEN GOTO EndOfRecordReached; END_IF;
END_REGION

REGION Network 61: **** 4.4 - Machine Status - Calculated **** Register Time events - OperatorOverCycle4 Start/stop
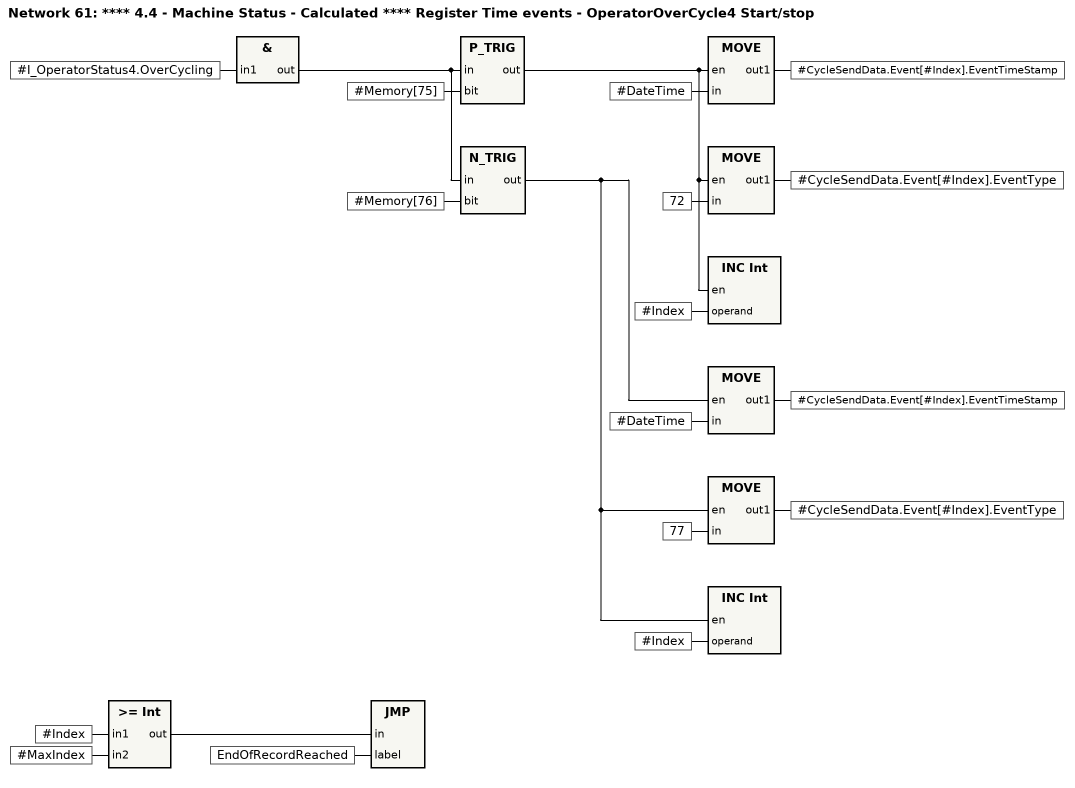
   #_w1 := #I_OperatorStatus4.OverCycling AND NOT #Memory[75];   // rising edge
   #Memory[75] := #I_OperatorStatus4.OverCycling;
   IF #_w1 THEN
       #CycleSendData.Event[#Index].EventTimeStamp := #DateTime;
       #CycleSendData.Event[#Index].EventType := 72;
       #Index := #Index + 1;
   END_IF;
   #_w2 := NOT #I_OperatorStatus4.OverCycling AND #Memory[76];   // falling edge
   #Memory[76] := #I_OperatorStatus4.OverCycling;
   IF #_w2 THEN
       #CycleSendData.Event[#Index].EventTimeStamp := #DateTime;
       #CycleSendData.Event[#Index].EventType := 77;
       #Index := #Index + 1;
   END_IF;
   IF #Index >= #MaxIndex THEN GOTO EndOfRecordReached; END_IF;
END_REGION

REGION Network 62: **** 4.4 - Machine Status - Calculated **** Register Time events - OperatorOverCycle5 Start/stop
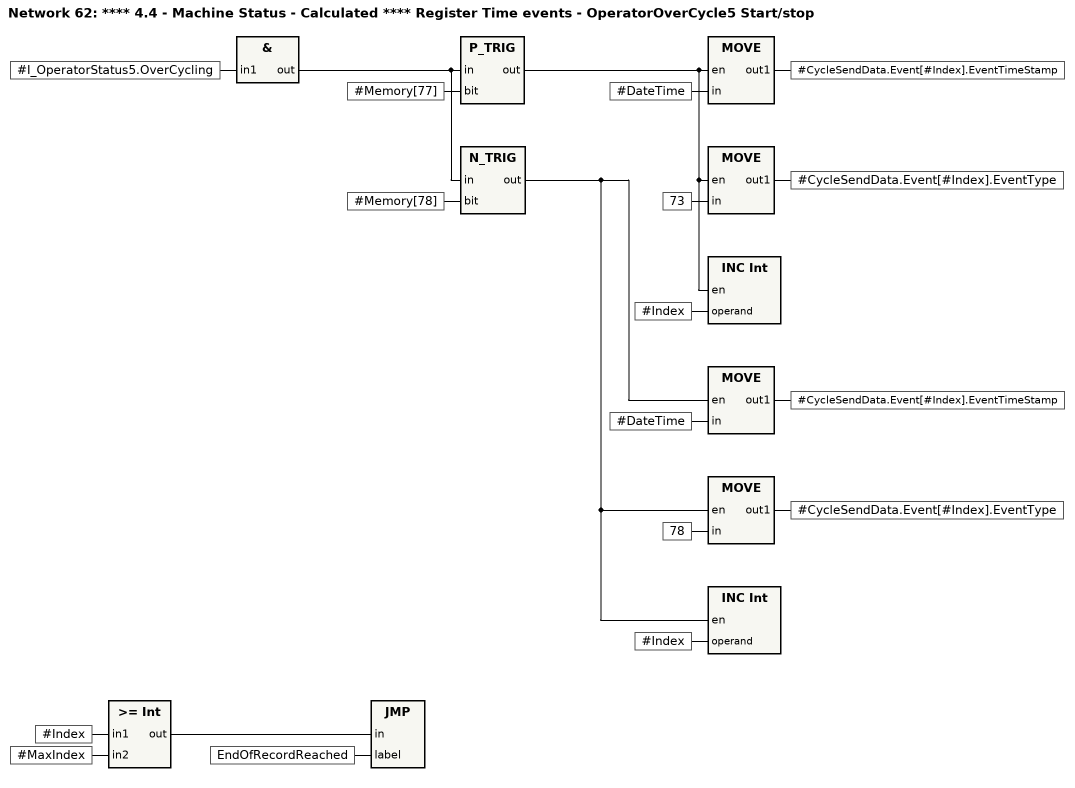
   #_w1 := #I_OperatorStatus5.OverCycling AND NOT #Memory[77];   // rising edge
   #Memory[77] := #I_OperatorStatus5.OverCycling;
   IF #_w1 THEN
       #CycleSendData.Event[#Index].EventTimeStamp := #DateTime;
       #CycleSendData.Event[#Index].EventType := 73;
       #Index := #Index + 1;
   END_IF;
   #_w2 := NOT #I_OperatorStatus5.OverCycling AND #Memory[78];   // falling edge
   #Memory[78] := #I_OperatorStatus5.OverCycling;
   IF #_w2 THEN
       #CycleSendData.Event[#Index].EventTimeStamp := #DateTime;
       #CycleSendData.Event[#Index].EventType := 78;
       #Index := #Index + 1;
   END_IF;
   IF #Index >= #MaxIndex THEN GOTO EndOfRecordReached; END_IF;
END_REGION

REGION Network 63: **** 4.4 - Machine Status - Calculated **** Register Time events - AutomaticOverCycle Start/stop
